
// ===== library: MasterCopy "Kopie von Programmbausteine in GW_Useranmeldung" =====

// folder: GW_Useranmeldung

DATA_BLOCK "DB Useranmeldung"   // DB42
{ S7_Optimized_Access := 'TRUE' }
VERSION : 0.1
   VAR
      HMI : "UDT_Useranmeldung";
      alive_send : Bool;
      alive_rcv : Bool;
      alive_fault : Bool;
   END_VAR
BEGIN
   HMI.local_user_name := 'user';
   HMI.local_user_pwd := '1111';
   HMI.local_user_access_level := 400;
   HMI.local_technician_name := 'service';
   HMI.local_technician_pwd := '2222';
   HMI.local_technician_access_level := 600;
   HMI.local_admin_name := 'admin';
   HMI.local_admin_pwd := '43194';
   HMI.local_admin_access_level := 1024;
   HMI.abmeldezeit := 600;
END_DATA_BLOCK

DATA_BLOCK "IDB_Useranmeldung"   // DB43
{ S7_Optimized_Access := 'TRUE' }
VERSION : 0.1
// stored: InstanceOfName FB_Useranmeldung
"FB_Useranmeldung"
BEGIN
END_DATA_BLOCK

DATA_BLOCK "IDB_AliveSystem"   // DB108
{ S7_Optimized_Access := 'TRUE' }
VERSION : 0.1
// stored: InstanceOfName FB_AliveSystem
"FB_AliveSystem"
BEGIN
END_DATA_BLOCK

FUNCTION_BLOCK "FB_Useranmeldung"   // FB38, FBD
{ S7_Optimized_Access := 'TRUE' }
VERSION : 0.1
   VAR
      max_time_login : TON_TIME;
      time_logout : TON_TIME;
   END_VAR
BEGIN

REGION Network 1
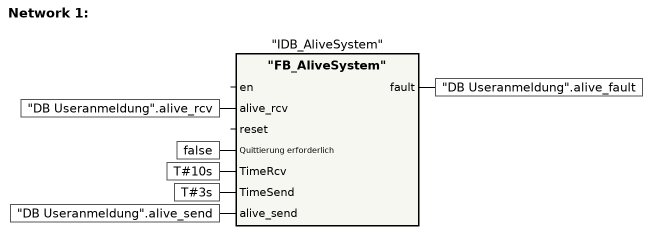
   "IDB_AliveSystem"(alive_rcv := "DB Useranmeldung".alive_rcv,   // "FB_AliveSystem"
                     "Quittierung erforderlich" := false,
                     TimeRcv := T#10s,
                     TimeSend := T#3s,
                     alive_send := "DB Useranmeldung".alive_send,
                     fault => "DB Useranmeldung".alive_fault);
END_REGION

REGION Network 2 (SCL): User Verwaltung lokal
   IF "DB Useranmeldung".HMI.check_local_input_trigger THEN

       IF "DB Useranmeldung".HMI.user_name_input = "DB Useranmeldung".HMI.local_user_name AND
           "DB Useranmeldung".HMI.pwd_input = "DB Useranmeldung".HMI.local_user_pwd THEN

           "DB Useranmeldung".HMI.active_user := "DB Useranmeldung".HMI.user_name_input;
           "DB Useranmeldung".HMI.access_level := "DB Useranmeldung".HMI.local_user_access_level;
       ELSIF
           "DB Useranmeldung".HMI.user_name_input = "DB Useranmeldung".HMI.local_technician_name AND
           "DB Useranmeldung".HMI.pwd_input = "DB Useranmeldung".HMI.local_technician_pwd THEN

           "DB Useranmeldung".HMI.active_user := "DB Useranmeldung".HMI.user_name_input;
           "DB Useranmeldung".HMI.access_level := "DB Useranmeldung".HMI.local_technician_access_level;
       ELSIF
           "DB Useranmeldung".HMI.user_name_input = "DB Useranmeldung".HMI.local_admin_name AND
           "DB Useranmeldung".HMI.pwd_input = "DB Useranmeldung".HMI.local_admin_pwd THEN

           "DB Useranmeldung".HMI.active_user := "DB Useranmeldung".HMI.user_name_input;
           "DB Useranmeldung".HMI.access_level := "DB Useranmeldung".HMI.local_admin_access_level;
      ELSE
          "DB Useranmeldung".HMI.active_user := '';
          "DB Useranmeldung".HMI.access_level := 0;
       END_IF;

      "DB Useranmeldung".HMI.check_local_input_trigger := FALSE;
      "DB Useranmeldung".HMI.user_name_input := '';
      "DB Useranmeldung".HMI.pwd_input := '';

   END_IF;
END_REGION

REGION Network 3 (SCL): User Verwaltung über Schnittstelle
   //Max.zeit für Login
   #max_time_login(IN := "DB Useranmeldung".HMI.check_input_trigger,
                   PT := T#5s);



   IF "DB Useranmeldung".HMI.login_user_trigger THEN
       "DB Useranmeldung".HMI.login_user_trigger := FALSE;
       "DB Useranmeldung".HMI.user_name_input := '';
       "DB Useranmeldung".HMI.pwd_input := '';
       "DB Useranmeldung".HMI.chip_id_input := '';
   END_IF;






   IF "DB Useranmeldung".HMI.check_input_trigger AND "DB Useranmeldung".HMI.access_level <> 0 THEN
       "DB Useranmeldung".HMI.chip_id_input := '';
   END_IF;




   IF #max_time_login.Q THEN
       "DB Useranmeldung".HMI.check_input_trigger := FALSE;
       "DB Useranmeldung".HMI.login_user_trigger := FALSE;
       "DB Useranmeldung".HMI.user_name_input := '';
       "DB Useranmeldung".HMI.pwd_input := '';
       "DB Useranmeldung".HMI.chip_id_input := '';
       "DB Useranmeldung".HMI.access_level := 0;


   END_IF;
END_REGION

REGION Network 4 (SCL): Abmeldezeit

   #time_logout(IN := "DB Useranmeldung".HMI.access_level > 1,
                PT := ("DB Useranmeldung".HMI.abmeldezeit * 1000));

   IF (#time_logout.Q OR "DB Useranmeldung".HMI.logout) THEN

       IF "DB Useranmeldung".HMI.startbildanwahl = TRUE THEN
           "DB Useranmeldung".HMI.startbildanwahl := FALSE;
       ELSE
           "DB Useranmeldung".HMI.startbildanwahl := TRUE;
       END_IF;

       "DB Useranmeldung".HMI.active_user := '';
       "DB Useranmeldung".HMI.user_name_input := '';
       "DB Useranmeldung".HMI.pwd_input := '';
       "DB Useranmeldung".HMI.chip_id_input := '';
       "DB Useranmeldung".HMI.access_level := 0;
       "DB Useranmeldung".HMI.logout := FALSE;
   END_IF;
END_REGION

REGION Network 5 (SCL)
   "DB Useranmeldung".HMI.verberge_popup := "DB Useranmeldung".HMI.access_level;

   IF "DB Useranmeldung".HMI.access_level < 0 THEN
       "DB Useranmeldung".HMI.login_fault := 1;
   ELSE
       "DB Useranmeldung".HMI.login_fault := 0;
   END_IF;
END_REGION
END_FUNCTION_BLOCK

FUNCTION_BLOCK "FB_AliveSystem"   // FB39, FBD
{ S7_Optimized_Access := 'TRUE' }
VERSION : 0.1
   VAR_INPUT
      alive_rcv : Bool;
      reset : Bool;
      "Quittierung erforderlich" : Bool;
      TimeRcv : Time;
      TimeSend : Time;
   END_VAR
   VAR_OUTPUT
      fault : Bool;
   END_VAR
   VAR_IN_OUT
      alive_send : Bool;
   END_VAR
   VAR
      quitt : Bool;
      "Timer.TonRcvOn" : TON_TIME;
      "Timer.TonRcvOff" : TON_TIME;
      "Timer.TonSendOn" : TON_TIME;
      "Timer.TpSendOff" : TP_TIME;
   END_VAR
   VAR_TEMP
      TON_DN : Bool;
      TOF_Dn : Bool;
      alive_send_tmp : Bool;
   END_VAR
BEGIN

REGION Network 1: Alive On Timer
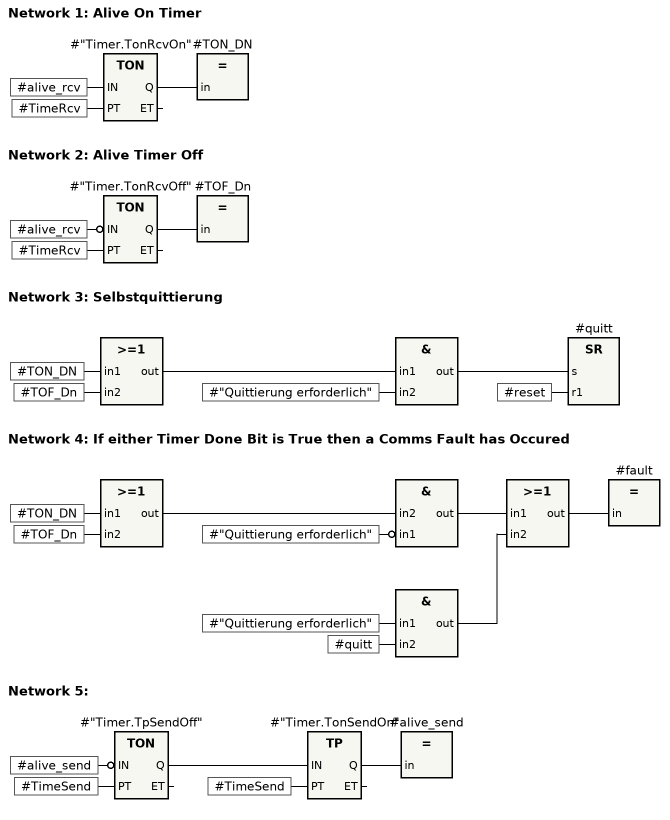
   #"Timer.TonRcvOn"(IN := #alive_rcv, PT := #TimeRcv);   // TON
   #TON_DN := #"Timer.TonRcvOn".Q;
END_REGION

REGION Network 2: Alive Timer Off
   #"Timer.TonRcvOff"(IN := NOT #alive_rcv, PT := #TimeRcv);   // TON
   #TOF_Dn := #"Timer.TonRcvOff".Q;
END_REGION

REGION Network 3: Selbstquittierung
   IF (#TON_DN OR #TOF_Dn) AND #"Quittierung erforderlich" THEN
       #quitt := TRUE;   // SR flip-flop
   END_IF;
   IF #reset THEN #quitt := FALSE; END_IF;
END_REGION

REGION Network 4: If either Timer Done Bit is True then a Comms Fault has Occured
   #fault := ((#TON_DN OR #TOF_Dn) AND NOT #"Quittierung erforderlich") OR (#"Quittierung erforderlich" AND #quitt);
END_REGION

REGION Network 5
   #"Timer.TpSendOff"(IN := NOT #alive_send, PT := #TimeSend);   // TON
   #"Timer.TonSendOn"(IN := #"Timer.TpSendOff".Q, PT := #TimeSend);   // TP
   #alive_send := #"Timer.TonSendOn".Q;
END_REGION
END_FUNCTION_BLOCK

// ===== library: MasterCopy "UDT_Useranmeldung" =====

TYPE "UDT_Useranmeldung"
   STRUCT
      user_name_input : String;
      pwd_input : String;
      chip_id_input : String;
      access_level : Int;
      active_user : String;
      check_input_trigger : Bool;
      check_local_input_trigger : Bool;
      login_user_trigger : Bool;
      local_user_name : String := 'user';
      local_user_pwd : String := '1111';
      local_user_access_level : Int := 400;
      local_technician_name : String := 'service';
      local_technician_pwd : String := '2222';
      local_technician_access_level : Int := 600;
      local_admin_name : String := 'admin';
      local_admin_pwd : String := '43194';
      local_admin_access_level : Int := 1024;
      verberge_popup : Int;
      startbildanwahl : Bool;
      logout : Bool;
      abmeldezeit : DInt := 600;
      login_fault : Bool;
   END_STRUCT;
END_TYPE

(* ===== HMI "HMI_RT_1" =====
system functions are stored by id; their names below are inferred from use

screen "Useranmeldung" 800x480
   TextField "Textfeld_1" at 259,116 size 315x30; Text 'Benutzeranmeldung'
   TextField "Textfeld_2" at 269,233 size 60x28; Text 'Login'
   TextField "Textfeld_3" at 268,367 size 74x28; Text 'Logout'
   TextField "Textfeld_4" at 269,276 size 45x22; Text 'User:'
   TextField "Textfeld_5" at 269,315 size 80x22; Text 'Passwort:'
   TextField "Textfeld_6" at 381,147 size 61x22; Text 'ChipID:'
   IOField "EA-Feld_2" at 355,311 size 210x30; FormatPattern ????????????????????????????????????????????????????????????????????????????????
      ProcessValue <- "DB Useranmeldung_HMI_pwd_input"
   IOField "EA-Feld_1" at 355,274 size 210x30; FormatPattern ????????????????????????????????????????????????????????????????????????????????
      ProcessValue <- "DB Useranmeldung_HMI_user_name_input"
   Button "Schaltfläche_3" at 354,366 size 210x30; TextOff 'Logout'
      on Activate: SetBit("DB Useranmeldung_HMI_logout")
      on Release: function_efd93a16()
   IOField "EA-Feld_5" at 268,174 size 296x30; FormatPattern ????????????????????????????????????????????????????????????????????????????????
      on OnFinishInput: function_efd93a16("Useranmeldung_1", 0, 0, 0, -1, 1)
      ProcessValue <- "DB Useranmeldung_HMI_chip_id_input"
   Button "Schaltfläche_1" at 525,117 size 47x28; TextOff 'X'
      on Press: function_efd93a16()
   Button "Schaltfläche_5" at 354,231 size 210x30; TextOff 'lokale Anmeldung'
      on Release: function_efd93a16()
      on Press: SetBit("DB Useranmeldung_HMI_check_local_input_trigger")
      Visibility <- "DB Useranmeldung_alive_fault"
   Button "Schaltfläche_2" at 354,231 size 210x30; TextOff 'Check'
      on Release: function_efd93a16()
      on Press: SetBit("DB Useranmeldung_HMI_check_input_trigger")
      Visibility <- "DB Useranmeldung_alive_fault"
   Button "Schaltfläche_4" at 354,231 size 210x30; TextOff 'Text'
      on Click: ActivateScreen("Useranmeldung_1", 0)
      Visibility <- "DB Useranmeldung_HMI_access_level"
*)